Staubli VAL3: IF.pjx

--- IF.pjx ---
Parameters version=s7.3.1 stackSize=5000 millimeterUnit=true
Program file=checkIn.pgx
Program file=checkOut.pgx
Program file=find.pgx
Program file=get.pgx
Program file=getPath.pgx
Program file=getSize.pgx
Program file=getType.pgx
Program file=insertCount.pgx
Program file=itemList.pgx
Program file=load.pgx
Program file=loadPage.pgx
Program file=onEdit.pgx
Program file=onInsert.pgx
Program file=onInsert_out.pgx
Program file=onProgEnd.pgx
Program file=onRun.pgx
Program file=onStart.pgx
Program file=onStop.pgx
Program file=showItem.pgx
Data file=IF.dtx
Library alias=cycleStatus path=Disk://cycleStatus/cycleStatus.pjx
Library alias=input path=Disk://instruction/inputOutput/IN/IN.pjx
Library alias=output path=Disk://instruction/inputOutput/OUT/OUT.pjx
Library alias=use path=Disk://kernel/userPage/userPage.pjx
Library alias=language path=Disk://kernel/language/language.pjx
Library alias=page path=Disk://kernel/template/page/page.pjx
Library alias=saveData path=Disk://saveData/saveData.pjx
Library alias=instruction path=Disk://..//templates/instruction/instruction.pjx
Library alias=language2 path=Disk://instruction/IF/language/language.pjx
Library alias=saveInOut path=Disk://saveInputOutput/saveInputOutput.pjx
Library alias=NUM path=Disk://instruction/inputOutput/NUM/NUM.pjx
Type name=InstrItem path=Disk://kernel/template/InstrItem/InstrItem.pjx
Type name=dioItem path=Disk://kernel/template/dioItem/dioItem.pjx

--- IF.dtx ---
string sChoice[4]
  [0] = "IN"
  [1] = "OUT"
  [3] = "NUM"
public string sItems
string sMessage

--- checkIn.pgx ---
program checkIn(string x_sItem (dimensions=1), bool& x_bResult[] (dimensions=1))
  local bool l_bMode[3]
  local string l_sItem[3]
  local num l_nCount
  local num l_nFlag
  local bool l_bActive
  local bool l_bFound
  local num l_nSize
  local num i
  local num j
  local string l_sName
  local string l_sMode
  local bool l_bStatus[3]
begin
  x_bResult=false
  //
  // find how many time and fill sItem and l_bMode
  //
  l_nCount=-1
  do
    l_nCount=l_nCount+1
    // l_sMode
    i=find(x_sItem,"AND")
    if i==-1
      i=find(x_sItem,"OR")
      if i!=-1
        l_sMode="OR"
        i=i+len("OR")+1
      endIf
    else
      l_sMode="AND"
      i=i+len("AND")+1
    endIf
    //
    if i!=-1
      l_sItem[l_nCount]=left(x_sItem,i)
      x_sItem=right(x_sItem,len(x_sItem)-i)
    else
      l_sItem[l_nCount]=x_sItem
    endIf
    l_nFlag=find(l_sItem[l_nCount],">")
    // l_bMode
    if find(l_sItem[l_nCount],">ON")!=-1
      l_bMode[l_nCount]=true
    else
      l_bMode[l_nCount]=false
    endIf
    //sItem
    l_sItem[l_nCount]=left(l_sItem[l_nCount],l_nFlag)
  until i==-1
  //
  call input:getStatus(l_bStatus,l_sItem[0])
  if l_sMode==""
    if (l_bStatus[0]==l_bMode[0])
      x_bResult=true
    endIf
  else
    // more then on event
    call input:getStatus(l_bStatus[1],l_sItem[1])
    //
    if l_sMode=="OR"
      switch l_nCount
        case 1
          if (l_bStatus[0]==l_bMode[0] or l_bStatus[1]==l_bMode[1])
            x_bResult=true
          endIf
        break
        case 2
          call input:getStatus(l_bStatus[2],l_sItem[2])
          if (l_bStatus[0]==l_bMode[0] or l_bStatus[1]==l_bMode[1] or l_bStatus[2]==l_bMode[2])
            x_bResult=true
          endIf
        break
      endSwitch
    else
      if l_sMode=="AND"
        switch l_nCount
          case 1
            if (l_bStatus[0]==l_bMode[0] and l_bStatus[1]==l_bMode[1])
              x_bResult=true
            endIf
          break
          case 2
            call input:getStatus(l_bStatus[2],l_sItem[2])
            if (l_bStatus[0]==l_bMode[0] and l_bStatus[1]==l_bMode[1] and l_bStatus[2]==l_bMode[2])
              x_bResult=true
            endIf
          break
        endSwitch
      endIf
    endIf
  endIf
end

--- checkOut.pgx ---
program checkOut(string x_sItem (dimensions=1), bool& x_bResult[] (dimensions=1))
  local bool l_bMode[3]
  local string l_sItem[3]
  local num l_nCount
  local num l_nFlag
  local bool l_bActive
  local bool l_bFound
  local num l_nSize
  local num i
  local num j
  local string l_sName
  local string l_sMode
  local bool l_bStatus[3]
begin
  x_bResult=false
  //
  // find how many time and fill sItem and l_bMode
  //
  l_nCount=-1
  do
    l_nCount=l_nCount+1
    // l_sMode
    i=find(x_sItem,"AND")
    if i==-1
      i=find(x_sItem,"OR")
      if i!=-1
        l_sMode="OR"
        i=i+len("OR")+1
      endIf
    else
      l_sMode="AND"
      i=i+len("AND")+1
    endIf
    //
    if i!=-1
      l_sItem[l_nCount]=left(x_sItem,i)
      x_sItem=right(x_sItem,len(x_sItem)-i)
    else
      l_sItem[l_nCount]=x_sItem
    endIf
    l_nFlag=find(l_sItem[l_nCount],">")
    // l_bMode
    if find(l_sItem[l_nCount],">ON")!=-1
      l_bMode[l_nCount]=true
    else
      l_bMode[l_nCount]=false
    endIf
    //sItem
    l_sItem[l_nCount]=left(l_sItem[l_nCount],l_nFlag)
  until i==-1
  //
  call output:getStatus(l_bStatus,l_sItem[0])
  if l_sMode==""
    if (l_bStatus[0]==l_bMode[0])
      x_bResult=true
    endIf
  else
    // more then on event
    call output:getStatus(l_bStatus[1],l_sItem[1])
    //
    if l_sMode=="OR"
      switch l_nCount
        case 1
          if (l_bStatus[0]==l_bMode[0] or l_bStatus[1]==l_bMode[1])
            x_bResult=true
          endIf
        break
        case 2
          call output:getStatus(l_bStatus[2],l_sItem[2])
          if (l_bStatus[0]==l_bMode[0] or l_bStatus[1]==l_bMode[1] or l_bStatus[2]==l_bMode[2])
            x_bResult=true
          endIf
        break
      endSwitch
    else
      if l_sMode=="AND"
        switch l_nCount
          case 1
            if (l_bStatus[0]==l_bMode[0] and l_bStatus[1]==l_bMode[1])
              x_bResult=true
            endIf
          break
          case 2
            call output:getStatus(l_bStatus[2],l_sItem[2])
            if (l_bStatus[0]==l_bMode[0] and l_bStatus[1]==l_bMode[1] and l_bStatus[2]==l_bMode[2])
              x_bResult=true
            endIf
          break
        endSwitch
      endIf
    endIf
  endIf
end

--- find.pgx ---
public program find(string& x_sItem[] (dimensions=1), bool& x_bFound[] (dimensions=1))
begin
end

--- get.pgx ---
public program get(string& x_sItem[] (dimensions=1), num x_nIndex (dimensions=1))
begin
end

--- getPath.pgx ---
program getPath(string& x_sType[] (dimensions=1))
  local num l_nPos
  local string l_sPath
  local num i
begin
  // get the TypePath
  call saveData:getPathInstr(x_sType,x_sType)
end

--- getSize.pgx ---
public program getSize(num& x_nSize[] (dimensions=1))
begin
end

--- insertCount.pgx ---
public program insertCount(string& x_sItem[])
  local num l_nSizeList
  local string l_sItem
  local num l_nSize
  local string l_sItemList
  local num l_nIndex
  local num i
  local num l_nValue
  local bool l_bActive
  local string l_sMessage
  local num l_nKey
  local string l_sEvent
  local string l_sEmpty
  local num l_nMode
  local string l_sButton[2]
  local bool l_bYes
begin
  cls()
  x_sItem=""
  // COUNT
  call NUM:getSize(l_nSizeList)
  l_sItem="NUM "
  l_nSize=0
  //
  // create the list
  //
  call use:setSizeList(21,0,17,10)
  call use:listcreate(l_sItem)
  // insert in the list
  for i=0 to l_nSizeList-1
    call NUM:get(l_sItemList,i)
    call NUM:isActive(l_bActive,l_sItemList)
    if l_bActive
      call use:listadd(l_sItemList)
    endIf
  endFor
  call use:listredraw(0)
  // display the actual item
  call use:type(2,12,l_sItem)
  call use:clear(0,13)
  call language:message(l_sMessage,63)
  call use:typeCenter(13,l_sMessage,40,true)
  do
    // get the key
    l_nKey=get()
    // get one input from the list
    call use:listevent(l_nKey,l_nIndex,l_sEvent)
    if l_nKey==255
      return
    endIf
  until l_nKey==270
  // check if an item has been selected
  if l_sEvent==""
    return
  endIf
  // compose the instruction
  x_sItem=l_sItem+l_sEvent
  // display the actual item
  call use:type(2,12,x_sItem)
  // Select the operator
  call language:message(l_sMessage,110)
  call use:questionDialog(l_sMessage,saveInOut:sOperator,i)
  // compose the istruction
  if i>=1 and i<=size(saveInOut:sOperator)
    x_sItem=x_sItem+saveInOut:sOperator[i-1]
  else
    // escape
    x_sItem=""
    return
  endIf
  // modify the actual item
  call use:type(2,12,x_sItem)
  // insert a value
  call language:message(l_sMessage,112)
  // get the yes_no button Key
  call language:getYesNo(l_sButton)
  // ask the question
  call use:yes_no(l_sMessage,l_sButton,l_bYes)
  // check it
  if l_bYes
    //
    // reuse the operator
    //
    // create the list
    call NUM:getSize(l_nSizeList)
    call getType(l_sItem)
    call use:setSizeList(21,0,17,10)
    call use:listcreate(l_sItem)
    // insert in the list
    for i=0 to l_nSizeList-1
      call NUM:get(l_sItemList,i)
      call NUM:isActive(l_bActive,l_sItemList)
      if l_bActive
        call use:listadd(l_sItemList)
      endIf
    endFor
    call use:listredraw(0)
    do
      // get the key
      l_nKey=get()
      // get one input from the list
      call use:listevent(l_nKey,l_nIndex,l_sEvent)
      if l_nKey==255
        return
      endIf
    until l_nKey==270
    // check if an item has been selected
    if l_sEvent==""
      x_sItem=""
      return
    else
      x_sItem=x_sItem+"NUM "+ l_sEvent
    endIf
  else
    // use a value
    call use:changeValue(l_nValue,-10000,10000,2+len(x_sItem),12,l_sEmpty)
    x_sItem=x_sItem+toString("",l_nValue)
  endIf
  // validate
  if use:bUseEscape
    x_sItem=""
  endIf
  //
end

--- itemList.pgx ---
program itemList(string& x_sEvent[])
  local num l_nSize
  local string l_sEvent
  local num l_nKey
  local num i
  local string l_sMessage
  local string l_sPath
  local num l_nResult
  local string l_sToto
begin
  //
  // USE this procedure to view the items
  // list that you have already save
  //
  cls()
  //
  if x_sEvent=="PROG"
    // Prog
    l_sPath="Disk://instruction/PROG"
  else
    // other
    l_sPath=x_sEvent
    call getPath(l_sPath)
  endIf
  // reload the instruction
  l_nResult=instruction:libLoad(l_sPath)
  delay(0)
  //
  if l_nResult==0
    //
    call instruction:onInsert(x_sEvent)
  else
    popUpMsg("error loading "+x_sEvent+" "+l_sPath+" "+toString("",l_nResult))
  endIf
end

--- onEdit.pgx ---
public program onEdit(string& x_sItem[] (dimensions=1))
  local string l_sItem
  local string l_sMessage
  local bool l_bContinue
  local string l_sProg
  local num l_nPos
  local num i
  local num l_nSize
  local string l_sPath
  local string l_sButton[2]
begin
  //
  // compose the string
  //
  call language2:getLanguage(l_sPath)
  if l_sPath!=language2:libPath()+"/"+saveData:language
    // set language
    call language2:setLanguage(language2:libPath()+"/"+saveData:language)
  endIf
  //
  l_nPos=find(x_sItem,"PROG")
  call getType(l_sItem)
  if size(x_sItem)>1
    if l_nPos!=-1
      call language2:message(l_sMessage,0)
      l_sProg=right(x_sItem,len(x_sItem)-l_nPos)
      // get the yes_no button Key
      call language:getYesNo(l_sButton)
      // ask the question
      call use:yes_no(l_sItem+" "+x_sItem+"##"+l_sMessage+"#"+l_sProg,l_sButton,l_bContinue)
      if l_bContinue
        x_sItem="Disk://instruction/PROG/page_viewInstr"
        x_sItem[1]=right(l_sProg,len(l_sProg)-len("PROG>"))
      endIf
    else
      popUpMsg(l_sItem+" "+x_sItem)
    endIf
  endIf
end

--- onInsert.pgx ---
public program onInsert(string& x_sItem[])
  local string l_sItem[5]
  local num l_nStep
  local num l_nResult
  local num l_nChoice
  local string l_sTemp
  local string l_sPath
  local string l_sMessage
  local string l_sType
  local num i
begin
  // get the language
  call language2:getLanguage(l_sPath)
  if l_sPath!=language2:libPath()+"/"+saveData:language
    // set language
    call language2:setLanguage(language2:libPath()+"/"+saveData:language)
  endIf
  call language2:message(l_sMessage,1)
  title(l_sMessage)
  for i=0 to size(l_sItem)-1
    l_sItem[i]=" "
  endFor
  // start how to insert
  while true
    cls()
    //
    // compose the string
    call getType(l_sType)
    call use:type(1,13,l_sType+" "+l_sItem+" "+l_sItem[1]+" "+l_sItem[2]+" "+l_sItem[3]+" "+l_sItem[4])
    switch l_nStep
      case -1
        x_sItem=""
        return
      break
      // SELECT FROM OUT/ IN / EMAP
      case 0
        call use:stringToArray("IN,OUT,,NUM",sChoice)
        call language2:message(l_sMessage,2)
        call use:questionDialog(l_sMessage,sChoice,l_nChoice)
        if l_nChoice>=1
          switch l_nChoice
            case 1
              l_sItem="IN"
            break
            case 2
              l_sItem="OUT"
            break
            //            case 3
            //              l_sItem="EMAP IN"
            //            break
            case 4
              l_sItem="NUM"
            break
          endSwitch
        else
          return
        endIf
        l_nStep=l_nStep+1
      break
      // SELECT FROM THE LIST
      case 1
        switch l_nChoice
          case 1
            call language2:message(l_sMessage,3)
            // insert the input from the list
            call input:onInsert(l_sItem[1])
          break
          case 2
            call language2:message(l_sMessage,4)
            // insert the input from the list
            call onInsert_out(l_sItem[1])
          break
          //          case 3
          //            call language2:message(l_sMessage,5)
          //            call use:type(1,11,l_sMessage)
          //            // insert the input from the list
          //            l_sItem[1]="IN"
          //            call euromap:onInsert(l_sItem[1])
          //          break
          case 4
            call language2:message(l_sMessage,4)
            // insert the input from the list
            l_sItem[1]="IF"
            call NUM:onInsert(l_sItem[1])
          break
        endSwitch
        //
        l_nStep=l_nStep+1
        //
      break
      case 2
        call use:stringToArray("CALL,GOTO",sChoice)
        call language2:message(l_sMessage,6)
        call use:questionDialog(l_sMessage,sChoice,l_nChoice)
        if l_nChoice==1 or l_nChoice==2
          switch l_nChoice
            case 1
              l_sItem[2]="CALL"
            break
            case 2
              l_sItem[2]="GOTO"
            break
          endSwitch
        endIf
        //
        l_nStep=l_nStep+1
        //
      break
      case 3
        // select the event
        call language2:message(l_sMessage,7)
        // show the list
        call showItem(l_sItem[3])
        //
        l_nStep=l_nStep+1
        //
      break
      case 4
        // seclect the item event
        call language2:message(l_sMessage,8)
        // show the item's list
        l_sItem[4]=l_sItem[3]
        call itemList(l_sItem[4])
        //
        l_nStep=l_nStep+1
        //
      break
      case 5
        // build the line
        if l_sItem!="" and l_sItem[1]!="" and l_sItem[2]!="" and l_sItem[3]!="" and l_sItem[4]!=""
          x_sItem=l_sItem+" "+l_sItem[1]+" "+l_sItem[2]+" "+l_sItem[3]+" "+l_sItem[4]
        else
          x_sItem=""
        endIf
        return
      break
    endSwitch
    //
    // step control
    //
    if l_nResult==-1 or l_sItem[1]=="" or l_sItem[2]=="" or l_sItem[3]==""
      l_nStep=-1
    endIf
  endWhile
end

--- onInsert_out.pgx ---
public program onInsert_out(string& x_sItem[])
  local num l_nSize
  local string l_sEvent
  local num i
  local num l_nKey
  local string l_sMessage
  local bool l_bActive
  local num l_nIndex
  local string l_sItemList
  local num l_nSizeList
  local string l_sButton[2]
  local string l_sKey
  local string l_sName
  local string l_sItem
begin
  x_sItem=""
  call getSize(l_nSizeList)
  do
    // create the list
    //
    call use:setSizeList(10,0,28,11)
    call use:listcreate("OUTPUT ")
    // start from the first
    l_sKey=first(saveInOut:dOutput)
    while l_sKey!=""
      // scan
      call output:isActive(l_bActive,l_sKey)
      if l_bActive
        // insert into the list
        l_sName=saveInOut:dOutput[l_sKey].sName
        l_sItemList=l_sKey+" {"+l_sName+"}"
        call use:listadd(l_sItemList)
      endIf
      // next
      l_sKey=next(saveInOut:dOutput[l_sKey])
    endWhile
    //
    // display the list
    //
    call use:listredraw(min(l_nIndex-use:nView,0))
    //
    // wait a KEY
    //
    do
      l_nKey=get()
      // get one input from the list
      call use:listevent(l_nKey,l_nIndex,l_sEvent)
      if l_nKey==255
        return
      endIf
    until l_nKey==270
    //
    // insert the sentence
    //
    if l_sEvent==""
      return
    else
      l_sEvent=left(l_sEvent,find(l_sEvent,"{")-1)
    endIf
    // update
    l_sItem=l_sItem+l_sEvent
    // get the status ON-OFF
    call use:stringToArray("ON,OFF",sMessage)
    call language:message(l_sMessage,40)
    call use:questionDialog(l_sMessage,sMessage,i)
    if i==1
      l_sItem=l_sItem+">ON"
    else
      if i==2
        l_sItem=l_sItem+">OFF"
      else
        // escape
        return
      endIf
    endIf
    l_nSize=l_nSize+1
    // define the operator
    if l_nSize!=3
      call language:message(l_sMessage,41)
      l_sButton="AND"
      l_sButton[1]="OR"
      call use:questionDialog(l_sMessage,l_sButton,i)
      if i==-1
        // escape
        return
      elseIf i==1
        l_sItem=l_sItem+" AND "
      elseIf i==2
        l_sItem=l_sItem+" OR "
      endIf
    endIf
  until i==0 or l_nSize==3
  // give it back
  x_sItem=l_sItem
end

--- onProgEnd.pgx ---
public program onProgEnd(string& x_sItem[] (dimensions=1))
begin
  //
  // Done, when one program has finished
  //
end

--- onRun.pgx ---
public program onRun(string& x_sItem[])
  local string l_sProg
  local num l_nPos
  local string l_sCondition
  local bool l_bCheck
  local num l_nType
  local string l_sItem
  local num l_nValue
  local num l_nOperator
  local num l_nIndex
begin
  //
  if find(x_sItem," GOTO")!=-1
    l_nType=0
    l_nPos=find(x_sItem," GOTO")
  else
    if find(x_sItem," CALL")!=-1
      l_nType=1
      l_nPos=find(x_sItem," CALL")
    endIf
  endIf
  // BUILD THE LINE
  l_sCondition=left(x_sItem,l_nPos)
  l_sItem=right(x_sItem,len(x_sItem)-l_nPos-len(" GOTO "))
  l_nPos=find(l_sItem," ")
  cycleStatus:sToShow=l_sItem
  // Decompose to iToSuperV
  if l_nPos!=-1
    cycleStatus:iToSuperV.sType=left(l_sItem,l_nPos)
    cycleStatus:iToSuperV.sData=right(l_sItem,len(l_sItem)-l_nPos-1)
  endIf
  // search the Input or Output*
  if find(left(l_sCondition,4),"IN ")!=-1
    // DISABLE THE INPUT LINE
    l_sCondition=right(l_sCondition,len(l_sCondition)-len(" IN"))
  elseIf find(left(l_sCondition,4),"OUT ")!=-1
    l_sCondition=right(l_sCondition,len(l_sCondition)-len(" OUT"))
    l_nType=l_nType+10
    //      elseIf find(left(l_sCondition,8),"EMAP IN ")!=-1
    //        l_sCondition=right(l_sCondition,len(l_sCondition)-len(" EMAP IN"))
    //        l_nType=l_nType+20
    //      endIf
  elseIf find(left(l_sCondition,6),"NUM ")!=-1
    l_sCondition=right(l_sCondition,len(l_sCondition)-len(" NUM"))
    l_nType=l_nType+30
  endIf
  //
  switch l_nType
    // GOTO INPUT
    case 0
      call checkIn(l_sCondition,l_bCheck)
      if l_bCheck
        // SET THE GOTO..
        cycleStatus:bGOTO=true
      endIf
    break
    // CALL INPUT
    case 1
      call checkIn(l_sCondition,l_bCheck)
      if l_bCheck
        // SET THE CALL..
        cycleStatus:bCALL=true
      endIf
    break
    // GOTO OUTPUT
    case 10
      call checkOut(l_sCondition,l_bCheck)
      if l_bCheck
        // SET THE GOTO..
        cycleStatus:bGOTO=true
      endIf
    break
    // CALL OUTPUT
    case 11
      call checkOut(l_sCondition,l_bCheck)
      if l_bCheck
        // SET THE CALL..
        cycleStatus:bCALL=true
      endIf
    break
    //    // GOTO EMAP IN
    //    case 20
    //      call checkEmapIn(l_sCondition,l_bCheck)
    //      if l_bCheck
    //        // SET THE GOTO..
    //        cycleStatus:bGOTO=true
    //      endIf
    //    break
    //    // CALL EMAP IN
    //    case 21
    //      call checkEmapIn(l_sCondition,l_bCheck)
    //      if l_bCheck
    //        // SET THE CALL..
    //        cycleStatus:bCALL=true
    //      endIf
    //    break
    // GOTO NUM
    case 30
      //...
      call saveInOut:decompose_wait(l_sCondition,l_sItem,l_nOperator,l_nValue)
      call NUM:condition(l_nOperator,l_nValue,l_sItem,l_bCheck)
      if l_bCheck
        // SET THE GOTO..
        cycleStatus:bGOTO=true
      endIf
    break
    // CALL NUM
    case 31
      //...
      call saveInOut:decompose_wait(l_sCondition,l_sItem,l_nOperator,l_nValue)
      call NUM:condition(l_nOperator,l_nValue,l_sItem,l_bCheck)
      if l_bCheck
        // SET THE CALL..
        cycleStatus:bCALL=true
      endIf
    break
  endSwitch
  // OK
  if l_bCheck
    // show the string
    use:bUseRefresh=true
  endIf
end

--- onStart.pgx ---
public program onStart(string& x_sItem[] (dimensions=1))
  local string l_sType
  local num i
  local string l_sPath
begin
  // language
  call language2:getLanguage(l_sPath)
  if l_sPath!=language2:libPath()+"/"+saveData:language
    // set language
    call language2:setLanguage(language2:libPath()+"/"+saveData:language)
  endIf
end

--- showItem.pgx ---
program showItem(string& x_sEvent[] (dimensions=1))
  local num l_nSize
  local string l_sEvent
  local num l_nKey
  local num i
  local string l_sMessage
begin
  //
  // USE this procedure to view Prog
  // that you have already saved
  //
  cls()
  call use:setView(false)
  //
  // Item list
  //
  call use:listcreate("")
  //
  l_nSize=size(saveData:sInstr)
  // refresh the list
  for i=0 to l_nSize-1
    l_sEvent=saveData:sInstr[i]
    if l_sEvent!="IF"
      call use:listadd(l_sEvent)
    endIf
  endFor
  call use:listupdate(0)
  call language:message(l_sMessage,60)
  call use:typeLen(0,13,l_sMessage,40)
  do
    l_nKey=get()
    call use:listevent(l_nKey,i,x_sEvent)
  until l_nKey==270 or l_nKey==255
  if l_nKey==255
    x_sEvent=""
  endIf
end
